PROGRAM IP2GEO_DEMO
VAR
	IP_C: IP_C;
	S_BUF: NETWORK_BUFFER;
	R_BUF: NETWORK_BUFFER;
	IP_CONTROL_1: IP_CONTROL;
	CLK_PRG : CLK_PRG;
	IP2GEO_1: IP2GEO;
	GEO: IP2GEO_DATA;
	activate: BOOL := TRUE;
	done: BOOL;
	busy: BOOL;
	error_c: DWORD;
	error_t: BYTE;
END_VAR
VAR // added by the converter: edge detectors and wires of the graphical bodies
    _w1 : ANY;
END_VAR

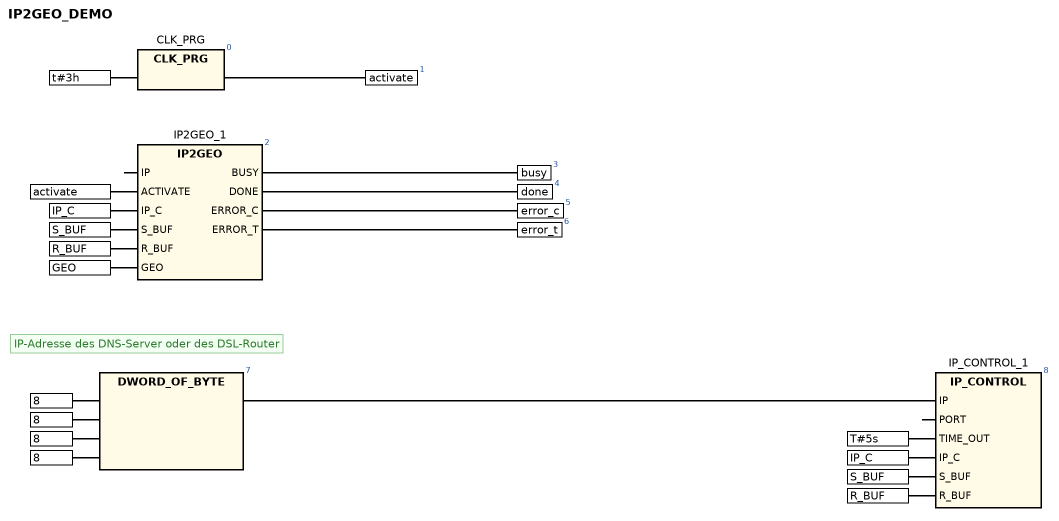
CLK_PRG(_in1 := t#3h);
activate := CLK_PRG._out1;
IP2GEO_1(ACTIVATE := activate, IP_C := IP_C, S_BUF := S_BUF, R_BUF := R_BUF, GEO := GEO); // IP2GEO
busy := IP2GEO_1.BUSY;
done := IP2GEO_1.DONE;
error_c := IP2GEO_1.ERROR_C;
error_t := IP2GEO_1.ERROR_T;
// IP-Adresse des DNS-Server oder des DSL-Router
_w1 := DWORD_OF_BYTE(8, 8, 8, 8);
IP_CONTROL_1(IP := _w1, TIME_OUT := T#5s, IP_C := IP_C, S_BUF := S_BUF, R_BUF := R_BUF); // IP_CONTROL

END_PROGRAM

(* stored: Version 1.1.0.1, ProductVersion 3.1.4024.9
   POU IP2GEO_DEMO: Id {45ded62d-c72f-42ce-acef-f9a4bd29abd0}, SpecialFunc None *)
